(*
SPDX-FileCopyrightText: Â© 2026 Oleksandr Tiutyk <trofimich@gmail.com>
SPDX-License-Identifier: MIT
License: https://opensource.org/license/mit
*)

(*!
<summary>Provides shared constants and metadata for automation controllers.</summary>
<description>
Supplies NoPlugins sentinel array for initializing controllers without extension plugins.
</description>
*)

{attribute 'no_explicit_call' := 'do not call this function block directly'}
PROGRAM AutomationControllers
VAR_OUTPUT CONSTANT
	(*! <summary>Empty array sentinel representing the absence of controller plugins.</summary> *)
	NoPlugins : ARRAY [0..-1] OF IAutomationControllerPlugin := [];
END_VAR
VAR
	_ClassName : STRING := __POUNAME();
END_VAR

(*!
<summary>Gets the class name of the program.</summary>
*)
{attribute 'monitoring' := 'call'}
PROPERTY ClassName : REFERENCE TO STRING
GET
ClassName REF= _ClassName;
END_GET
END_PROPERTY

(*!
<summary>Gets the namespace of the program.</summary>
*)
{attribute 'monitoring' := 'call'}
PROPERTY NamespaceName : REFERENCE TO STRING
GET
NamespaceName REF= CurrentNamespace.Name;
END_GET
END_PROPERTY

END_PROGRAM

(* stored: Version 1.1.0.1
   POU AutomationControllers: Id {3e9e98b1-6fa6-4b80-995a-c67a0fc3ee37}, SpecialFunc None
   Property ClassName: Id {da331e39-5c52-4d20-9e20-dc3ba2063c40}
   Get Get: Id {1da40aab-6580-4da9-bbb0-5ef1b5dd0c8e}
   Property NamespaceName: Id {b3b84c5c-106a-4842-ac2a-c8d0e507d7c1}
   Get Get: Id {ecb788f6-17b2-49f2-a08d-a24d1014fe27} *)
